//==================================================================================================
//							Beckhoff Automation Poland
//									30.03.2017
//	Proste zliczanie czasu pracy, podaje czas aktualnego zalaczenia, ostatniego zalaczenia, sumarycznego zalaczenia
// 	v1.0	|| TC v 3.1.4020.32		|| - pierwsza wersja
//==================================================================================================
FUNCTION_BLOCK FB_SimpleWorkTime
VAR_INPUT
	bIn										: BOOL;
	bReset									: BOOL;					// Zerowanie wartosci
END_VAR
VAR_OUTPUT
	tCurrentTime							: TIME;					// Aktualny czas zalaczenia
	tLastTime								: TIME;					// Ostatni czas zalaczenia
	tSummaryTime							: TIME;					// Sumaryczny czas zalaczenia
END_VAR
VAR
	fbTimeMeasure							: FB_TimeMeasureEx;		// Licznik czasu
	tLastSummaryTime						: TIME;					// Zmienna do wewnetrznych przeliczen
END_VAR

fbTimeMeasure(bOn:= bIn, bReset := bReset, tCurrentTime=> tCurrentTime, tLastTime=> tLastTime);
IF bIn THEN
	tSummaryTime 		:= tLastSummaryTime + tCurrentTime;
ELSE
	tLastSummaryTime 	:= tSummaryTime;
END_IF

IF bReset THEN
	tSummaryTime 		:= T#0S;
	tLastSummaryTime 	:= T#0S;
END_IF

END_FUNCTION_BLOCK

(* stored: Version 1.1.0.1, ProductVersion 3.1.4020.12
   POU FB_SimpleWorkTime: Id {c9a69df4-bfc4-40bd-8953-4fbbee48153c}, SpecialFunc None *)
